// TIA Portal V20 export
VAR_GLOBAL   // PLC tag table "LGR_Const_IO_ConfigID"
END_VAR
VAR_GLOBAL CONSTANT   // user constants
   IOCONFIG_RND : SInt := 0;
   IOCONFIG_INSFECTION_1 : SInt := 11;
   IOCONFIG_INBOUND_1 : SInt := 12;
   IOCONFIG_OUTBOUND_RETURN : SInt := 31;
   IOCONFIG_INSFECTION_2 : SInt := 21;
   IOCONFIG_INBOUND_2 : SInt := 22;
   IOCONFIG_TBR_INBOUND : SInt := 101;
   IOCONFIG_OUTBOUND_1 : SInt := 41;
   IOCONFIG_OUTBOUND_2 : SInt := 51;
   IOCONFIG_OUTBOUND_3 : SInt := 61;
END_VAR
